Staubli VAL3: clkDoTest.pgx

program clkDoTest()
begin
  bDoTest=true
end
